PROGRAM P_FastScan
VAR
	ID						:INT:=FastScan;
	SysStep:				DINT;	
	HomeStep:				DINT;	
	RestStep				:DINT;
	MoveStep				:DINT;
	HomeDone:               BOOL;
	FB_move:				FB_MoveFS_Exte;
	FB_home:				FB_Home_X;
	ton_commandtimeout		:TON;

	ton1:Tc2_Standard.TON;	//	命令延迟关闭
	Move_Done				:BOOL;
	NOT_Moving_TimeOut		:BOOL;
	parameter_out_of_range	:BOOL;
	actuator_out_of_pos_range:BOOL;
	actuator_out_of_neg_range:BOOL;	
	homeTimeOut				:BOOL;
	SpeedNotReach			:BOOL;	
	jog_EN					:BOOL;
	ton_Moving				:TON;
	
	direN:BOOL;
	direp:BOOL;
	log_ErrorEnum:Axis_XY_ErrorEnum;
	log_ID:INT;
	i:INT;
	
END_VAR

ACT_LOG();
GVL_API.stAxis[ID].ControlLoopClosed:=Axis[ID].Ref.Status .ControlLoopClosed;

(*****************POS******************************)
GVL_API.stAxis[ID].position:=Axis[ID].Ref.NcToPlc.ActPos;
direN:=Axis[ID].Ref.Status.NegativeDirection;
direp:=Axis[ID].Ref.Status.PositiveDirection;
(*****************SysStep******************************)
CASE SysStep OF
0:	(*wait*)
	_00_Waiting();				
100:(*idle*)		
	_100_Idle();								
200:(*home*)		
	_200_Homing();
300:(*ready*)	
	_300_Ready();							
400:(*disable*)	
	_400_Disable();			
500:(*Moving*)
	_500_Moving();	
600:(*Stopping*)
	_600_Stopping();
700:(*Error*)
	_700_Error();	
800:(*Reset*)
	_800_Reset();		
END_CASE

(*****************Reset*************************)
IF GVL_API.stAxis[ID].reset OR GVL.Reset THEN 
	SysStep:=800;	
END_IF

ACT_SAFETY();


Axis[ID].aReadStatus();
Axis[ID].aReset();

ACTION _00_Waiting:
IF GVL_API.stAxis[ID].initialize THEN 
	GVL_API.stAxis[ID].initialize:=FALSE;
	Axis[ID].aStop(stop_do:=TRUE);
	SysStep:=100;
ELSIF GVL_API.stAxis[ID].homeExe THEN 
	GVL_API.stAxis[ID].homeExe:=FALSE;  
	GVL_API.stAxis[ID].Home_Done:=FALSE;
	SysStep:=200;
ELSIF GVL_API.stAxis[ID].MoveAbsoluteExe OR GVL_API.stAxis[ID].MoveRelativeExe 
		OR GVL_API.stAxis[ID].MoveVelocityExe OR GVL_API.stAxis[ID].JogBackwards 
		OR GVL_API.stAxis[ID].JogForward OR GVL_API.stAxis[ID].MoveConstantVelocity
		OR GVL_API.stAxis[ID].enabled OR GVL_API.stAxis[ID].Disable THEN 
	GVL_API.stAxis[ID].Move_Done:=FALSE;
	SysStep:=300;	
ELSIF GVL_API.stAxis[ID].stop THEN 
	SysStep:=600;	
ELSIF GVL_API.stAxis[ID].reset OR GVL.Reset THEN 
	SysStep:=800;	
END_IF

ton1(IN:=GVL_API.stAxis[ID].Home_Done OR  GVL_API.stAxis[ID].Move_Done , PT:=State_reset_time , Q=> , ET=> );
IF ton1.Q THEN 
	GVL_API.stAxis[ID].Home_Done:=FALSE;
	GVL_API.stAxis[ID].Move_Done:=FALSE;
END_IF
END_ACTION

ACTION _100_Idle:
Axis[ID].aStop(stop_do:=FALSE);
Axis[ID].aPower(power_do:=TRUE);	

IF axis[Id].Ref.Status .ControlLoopClosed THEN 
	GVL_API.stAxis[ID].state:=AxisStateEnum.idle;
	SysStep :=0;
ELSIF GVl.Emstop_Button OR GVL.Emstop_SAFE THEN 
	GVL_API.stAxis[ID].errorid:=Axis_XY_ErrorEnum.emergency_error;
	SysStep:=700;
END_IF

(*******************commandtimeout*********************************)
ton_commandtimeout(IN:=NOT axis[Id].Ref.Status .ControlLoopClosed , 
	PT:=LREAL_TO_TIME(GVL_API.stAxis[ID].commandtimeout*1000) ,
	Q=> , ET=> );
IF ton_commandtimeout.Q  THEN 
	ton_commandtimeout(IN:=FALSE );
	GVL_API.stAxis[ID].errorid:=Axis_XY_ErrorEnum.cmd_timeout;
	SysStep:=700;	
END_IF

(*****************RESET******************************)
IF GVL_API.stAxis[ID].reset OR GVL.HMI_btReset   THEN
	 SysStep:=800;
END_IF
END_ACTION

ACTION _200_Homing:
FB_Home(
		ref:=				Axis[ID].Ref , 
		Execute:= , 
		PosLimit:=			Axis[ID].IO.snLimitP , 
		Position:=			0 , 
		HomeingVelo:=		GVL_API.stAxis[ID].homingvelocity , 
		Standby_position:=  GVL_API.stAxis[ID].homeoffset,
		bCalibrationCam:=	Axis[ID].IO.snHome , 
		rel_dis:=			50 , 
		TimeOutSet:=		GVL_API.stAxis[ID].homingtimeout , 
		reset:= , 
		Done=> , 
		Busy=> , 
		Active=> , 
		CommandAborted=> , 
		Error=> , 
		ErrorID=> , 
		TimeOut=> );
		
CASE HomeStep OF
0:
	IF GVL_API.stAxis[ID].homingvelocity<>0 THEN 
		HomeStep:=10;
	END_IF
10:
	FB_Home.Execute:=TRUE;					
	IF FB_Home.Done THEN
		GVL_API.stAxis[ID].Home_Done:=TRUE;
		FB_Home.Execute:=FALSE;		
		HomeStep:=20;
	END_IF
	IF FB_Home.Error THEN 		
		GVL_API.stAxis[ID].ErrorId:=Axis_XY_ErrorEnum.homing_timeout;
		HomeStep:=30;
	END_IF
	
20:	(**********HOME DONE****************)	
	GVL_API.stAxis[ID].state:=AxisStateEnum.ready;	
	HomeStep:=0;	
	SysStep:=0;
		
30:(**********TIME OUT****************)
	FB_Home.Execute:=FALSE;
	FB_Home.reset:=TRUE;
	HomeStep:=40;
40:(**********RESET****************)
	FB_Home.reset:=FALSE;
	HomeStep:=0;
	SysStep:=700;
		
END_CASE

IF FB_Home.Busy THEN 
	GVL_API.stAxis[ID].state:=AxisStateEnum.homing;
END_IF


(*****************RESET******************************)
IF GVL_API.stAxis[ID].reset    THEN
	FB_Home.Execute:=FALSE;
	 SysStep:=800;
END_IF
END_ACTION

ACTION _300_Ready:
Axis[ID].aStop();
GVL_API.stAxis[ID].Move_Done:=FALSE;
(***********parameter_out_of_range***********)
IF GVL_API.stAxis[ID].requestedposition>GVL_API.stAxis[ID].maxDistance OR GVL_API.stAxis[ID].requestedposition<0 THEN 
		parameter_out_of_range:=TRUE;
ELSIF GVL_API.stAxis[ID].constantvelocitystart>GVL_API.stAxis[ID].maxDistance OR GVL_API.stAxis[ID].constantvelocitystart<0 THEN
		parameter_out_of_range:=TRUE;
ELSIF GVL_API.stAxis[ID].constanvelocityend>GVL_API.stAxis[ID].maxDistance OR GVL_API.stAxis[ID].constanvelocityend<0 THEN
		parameter_out_of_range:=TRUE;	
ELSIF  GVL_API.stAxis[ID].requestedoffset>0 
	AND (GVL_API.stAxis[ID].maxDistance-Axis[ID].Ref.NcToPlc.ActPos)<GVL_API.stAxis[ID].requestedoffset THEN
	 	parameter_out_of_range:=TRUE;
ELSIF GVL_API.stAxis[ID].requestedoffset<-1	
	AND Axis[ID].Ref.NcToPlc.ActPos<ABS(GVL_API.stAxis[ID].requestedoffset) THEN 
		parameter_out_of_range:=TRUE;

ELSE
		parameter_out_of_range:=FALSE;
END_IF	

(*********out_of_pos_range****************)
IF Axis[ID].Ref.NcToPlc.ActPos>GVL_API.stAxis[ID].maxDistance THEN 
	actuator_out_of_pos_range:=TRUE;
	actuator_out_of_neg_range:=FALSE;		
ELSIF	Axis[ID].Ref.NcToPlc.ActPos<-1 THEN 
	actuator_out_of_pos_range:=FALSE;
	actuator_out_of_neg_range:=TRUE;
ELSE
	actuator_out_of_pos_range:=FALSE;
	actuator_out_of_neg_range:=FALSE;
END_IF
	

(*****************state******************************)
IF Axis[ID].Ref.Status.NotMoving AND axis[Id].Ref.Status .ControlLoopClosed  
AND NOT Axis[ID].Ref.Status.Error THEN 
	IF parameter_out_of_range THEN 
		GVL_API.stAxis[ID].errorid:=Axis_XY_ErrorEnum.parameter_out_of_range;
		SysStep:=700;
	ELSIF actuator_out_of_pos_range THEN 
		GVL_API.stAxis[ID].errorid:=Axis_XY_ErrorEnum.actuator_out_of_pos_range;
		SysStep:=700;
	ELSIF actuator_out_of_neg_range THEN 
		GVL_API.stAxis[ID].errorid:=Axis_XY_ErrorEnum.actuator_out_of_neg_range;
		SysStep:=700;	
	ELSE
		GVL_API.stAxis[ID].state:=AxisStateEnum.ready;
		GVL_API.stAxis[ID].errorid:=Axis_XY_ErrorEnum.no_error;
	END_IF
END_IF

(*****************valid command******************************)
IF NOT parameter_out_of_range 
AND axis[Id].Ref.Status .ControlLoopClosed  THEN  			
	IF GVL_API.stAxis[ID].MoveAbsoluteExe OR GVL_API.stAxis[ID].MoveRelativeExe 
		OR GVL_API.stAxis[ID].MoveVelocityExe OR GVL_API.stAxis[ID].JogBackwards 
		OR GVL_API.stAxis[ID].JogForward OR GVL_API.stAxis[ID].MoveConstantVelocity	THEN 	  		
			SysStep:=500;		
	END_IF
END_IF

(*****************enable-disable******************************)
IF GVL_API.stAxis[ID].enabled THEN 
	Axis[Id].aPower(power_do:=TRUE);	
	GVL_API.stAxis[ID].enabled:=FALSE;
	 GVL_API.stAxis[ID].state:=AxisStateEnum.ready;
	SysStep :=0;
ELSIF  GVL_API.stAxis[ID].Disable THEN 
	  SysStep:=400;
END_IF


(*****************RESET******************************)
IF GVL_API.stAxis[ID].reset THEN
	 SysStep:=800;
END_IF
END_ACTION

ACTION _400_Disable:
(*****************enable-disable******************************)
IF GVL_API.stAxis[ID].Disable THEN 
	Axis[Id].aPower(power_do:=FALSE);
	GVL_API.stAxis[ID].Disable:=FALSE;
	GVL_API.stAxis[ID].state:=AxisStateEnum.disabled;
	//IF NOT  axis[Id].Ref.Status .ControlLoopClosed THEN 
		SysStep:=0;
	//END_IF
	
END_IF

(*****************RESET******************************)
IF GVL_API.stAxis[ID].reset THEN
	 SysStep:=800;
END_IF
END_ACTION

ACTION _500_Moving:
GVL_API.stAxis[ID].state:=AxisStateEnum.moving;

(*********out_of_pos_range****************)
IF Axis[ID].Ref.NcToPlc.ActPos>GVL_API.stAxis[ID].maxDistance THEN 
	actuator_out_of_pos_range:=TRUE;
	actuator_out_of_neg_range:=FALSE;
	GVL_API.stAxis[ID].JogForward:=FALSE;		
ELSIF	Axis[ID].Ref.NcToPlc.ActPos<-1 THEN 
	actuator_out_of_pos_range:=FALSE;
	actuator_out_of_neg_range:=TRUE;
	GVL_API.stAxis[ID].JogBackwards:=FALSE;
ELSE
	actuator_out_of_pos_range:=FALSE;
	actuator_out_of_neg_range:=FALSE;
END_IF

(*********parameter_out_of_range****************)
IF Axis[ID].IO.snHome 
	AND (GVL_API.stAxis[ID].requestedoffset<0 
	OR GVL_API.stAxis[ID].constantvelocitystart<Axis[ID].Ref.NcToPlc.ActPos
	OR GVL_API.stAxis[ID].constanvelocityend<Axis[ID].Ref.NcToPlc.ActPos
	OR GVL_API.stAxis[ID].requestedposition<Axis[ID].Ref.NcToPlc.ActPos)
	THEN 	parameter_out_of_range:=TRUE;
ELSIF Axis[ID].IO.snLimitP
	AND (GVL_API.stAxis[ID].requestedoffset>0 
	OR GVL_API.stAxis[ID].constantvelocitystart>Axis[ID].Ref.NcToPlc.ActPos
	OR GVL_API.stAxis[ID].constanvelocityend>Axis[ID].Ref.NcToPlc.ActPos
	OR GVL_API.stAxis[ID].requestedposition>Axis[ID].Ref.NcToPlc.ActPos)
	THEN 	parameter_out_of_range:=TRUE;
END_IF


IF NOT_Moving_TimeOut OR GVL_API.stAxis[ID].Move_Done  THEN 			(************NOT_Moving_TimeOut/Move_Done**************)
	NOT_Moving_TimeOut:=FALSE;	
	GVL_API.stAxis[ID].state:=AxisStateEnum.ready;			
	SysStep:=0;
ELSIF SpeedNotReach THEN 							(************SpeedNotReach**************)
	GVL_API.stAxis[ID].errorid:=Axis_XY_ErrorEnum.SpeedNotReach;
	SysStep:=700;
ELSIF Axis[ID].Ref.Status.NotMoving AND parameter_out_of_range THEN 
	GVL_API.stAxis[ID].errorid:=Axis_XY_ErrorEnum.parameter_out_of_range;
	SysStep:=700;
ELSIF Axis[ID].Ref.Status.Moving THEN 				(************trigger_limit**************)
	IF (Axis[ID].Ref.Status.NegativeDirection AND Axis[ID].IO.snLimitN) OR 
		(Axis[ID].Ref.Status.PositiveDirection AND Axis[ID].IO.snLimitP) 
		OR stInput.biElectromagnet_limit  OR stOutput.bqElectromagnet_power 
	THEN	
		Axis[ID].aStop(stop_do:=TRUE);
		GVL_API.stAxis[ID].errorid:=Axis_XY_ErrorEnum.trigger_limit;
		SysStep:=700;	
	END_IF 
	
ELSIF actuator_out_of_pos_range THEN 					(*********out_of_pos_range****************)
	Axis[ID].aStop(stop_do:=TRUE);
	GVL_API.stAxis[ID].errorid:=Axis_XY_ErrorEnum.actuator_out_of_pos_range;
	SysStep:=700;
ELSIF actuator_out_of_neg_range THEN
	Axis[ID].aStop(stop_do:=TRUE); 
	GVL_API.stAxis[ID].errorid:=Axis_XY_ErrorEnum.actuator_out_of_neg_range;
	SysStep:=700;	
ELSE GVL_API.stAxis[ID].errorid:=Axis_XY_ErrorEnum.no_error;
END_IF


(*****************JOG/ABS/REL/******************************)
(*****************MoveConstantVelocity*****************************)
IF NOT parameter_out_of_range  THEN 
	FB_move(
	enable:= 					NOT stInput.biElectromagnet_limit AND NOT stOutput.bqElectromagnet_power,	
	ref:= 						Axis[ID].Ref, 
	jogF:= 						GVL_API.stAxis[ID].JogForward, 
	jogB:= 						GVL_API.stAxis[ID].JogBackwards, 
	Move_Stop:=				GVL_API.stAxis[ID].stop OR GVL_API.stAxis[ID].reset ,
	PosLimit:=					Axis[ID].IO.snLimitP , 
	NegLimit:= 					Axis[ID].IO.snLimitN, 
	maxDistance:=				GVL_API.stAxis[ID].maxDistance ,	
	Acceleration:= 				GVL_API.stAxis[ID].acceleration, 
	Deceleration:= 				GVL_API.stAxis[ID].acceleration, 
	Jerk:= 						GVL_API.stAxis[ID].jerk, 	 
	MoveRelExe:= 				GVL_API.stAxis[ID].MoveRelativeExe, 
	MoveAbsExe:= 				GVL_API.stAxis[ID].MoveAbsoluteExe, 
	MoveConstantVelocityExe:= 	GVL_API.stAxis[ID].MoveConstantVelocity, 
	Velo:= 						GVL_API.stAxis[ID].velocity, 
	TargetRel:= 				GVL_API.stAxis[ID].requestedoffset, 
	TargetAbs:= 				GVL_API.stAxis[ID].requestedposition, 
	constantvelocitystart:= 	GVL_API.stAxis[ID].constantvelocitystart, 
	constanvelocityend:= 		GVL_API.stAxis[ID].constanvelocityend, 
	Done:= 						GVL_API.stAxis[ID].Move_Done,
	NotMovingTimeOut:= 			NOT_Moving_TimeOut,
	SpeedNotReach:=				SpeedNotReach
	);	
END_IF


(*****************stop******************************)
IF GVL_API.stAxis[ID].stop THEN 
	SysStep:=600;
END_IF
(*****************RESET******************************)
IF GVL_API.stAxis[ID].reset THEN
	 SysStep:=800;
END_IF
END_ACTION

ACTION _600_Stopping:
(**************只单独用作STOP命令*************************)
GVL_API.stAxis[ID].state:=AxisStateEnum.stopping;

Axis[ID].aStop(stop_do:=GVL_API.stAxis[ID].stop,Jerk:=GVL_API.stAxis[ID].jerk);
IF Axis[ID].mcStop.Busy THEN 
	GVL_API.stAxis[ID].state:=AxisStateEnum.stopping;	
	GVL_API.stAxis[ID].JogBackwards:=FALSE;
	GVL_API.stAxis[ID].JogForward:=FALSE;
	GVL_API.stAxis[ID].MoveAbsoluteExe:=FALSE;
	GVL_API.stAxis[ID].MoveConstantVelocity:=FALSE;
	GVL_API.stAxis[ID].MoveRelativeExe:=FALSE;
	GVL_API.stAxis[ID].velocity:=0;
	GVL_API.stAxis[ID].requestedoffset:=0;
	GVL_API.stAxis[ID].requestedposition:=0;
	GVL_API.stAxis[ID].stop:=FALSE;
END_IF

IF Axis[ID].mcStop.Done AND Axis[ID].Ref.Status.NotMoving   THEN 		
	GVL_API.stAxis[ID].stop:=FALSE;
	GVL_API.stAxis[ID].state:=AxisStateEnum.ready;	
	GVL_API.stAxis[ID].Move_Done:=TRUE;
	SysStep:=0;
END_IF

(*****************RESET******************************)
IF GVL_API.stAxis[ID].reset THEN
	 GVL_API.stAxis[ID].stop:=FALSE;
	 Axis[ID].aStop(stop_do:=FALSE);
	 SysStep:=800;
END_IF
END_ACTION

ACTION _700_Error:
(*****************ERROR******************************)
GVL_API.stAxis[ID].Error:=TRUE;
GVL_API.stAxis[ID].state:=AxisStateEnum.error;
		GVL_API.stAxis[ID].initialize:=FALSE;
		GVL_API.stAxis[ID].homeExe:=FALSE; 
		GVL_API.stAxis[ID].stop:=FALSE;
		GVL_API.stAxis[ID].JogBackwards:=FALSE;
		GVL_API.stAxis[ID].JogForward:=FALSE;
		GVL_API.stAxis[ID].MoveAbsoluteExe:=FALSE;
		GVL_API.stAxis[ID].MoveConstantVelocity:=FALSE;
		GVL_API.stAxis[ID].MoveRelativeExe:=FALSE;
		GVL_API.stAxis[ID].velocity:=0;
		GVL_API.stAxis[ID].requestedoffset:=0;
		GVL_API.stAxis[ID].requestedposition:=0;
		GVL_API.stAxis[ID].constantvelocitystart:=0;
		GVL_API.stAxis[ID].constanvelocityend:=0;
		FB_Home.Execute:=FALSE;
		GVL_API.stAxis[ID].Home_Done:=FALSE;
		GVL_API.stAxis[ID].Move_Done:=FALSE;
 SysStep:=0;
END_ACTION

ACTION _800_Reset:
Axis[ID].aStop();
CASE RestStep OF
0:(***************复位命令**************************)
	IF GVL_API.stAxis[ID].reset OR GVL.Reset THEN
		GVL_API.stAxis[ID].initialize:=FALSE;
		GVL_API.stAxis[ID].homeExe:=FALSE; 
		GVL_API.stAxis[ID].stop:=FALSE;
		GVL_API.stAxis[ID].JogBackwards:=FALSE;
		GVL_API.stAxis[ID].JogForward:=FALSE;
		GVL_API.stAxis[ID].MoveAbsoluteExe:=FALSE;
		GVL_API.stAxis[ID].MoveConstantVelocity:=FALSE;
		GVL_API.stAxis[ID].MoveRelativeExe:=FALSE;
		GVL_API.stAxis[ID].velocity:=0;
		GVL_API.stAxis[ID].requestedoffset:=0;
		GVL_API.stAxis[ID].requestedposition:=0;
		GVL_API.stAxis[ID].constantvelocitystart:=0;
		GVL_API.stAxis[ID].constanvelocityend:=0;
		FB_Home(ref:=Axis[ID].Ref , Execute:= FALSE);
		GVL_API.stAxis[ID].Home_Done:=FALSE;
		GVL_API.stAxis[ID].Move_Done:=FALSE;
		RestStep:=1;
	END_IF
1:	
		RestStep:=2;

2:(***************EORROR来的错误**************************)
		GVL_API.stAxis[ID].reset:=FALSE;
		parameter_out_of_range:=FALSE;
		SpeedNotReach:=FALSE;		
		RestStep:=20;
	
10:	(***************轴错误复位**************************)		
		Axis[ID].Reset_do:=TRUE;		
		RestStep:=100;		
20:	(***************轴停止*****************************)
		Axis[ID].aStop(stop_do:=TRUE);		
		RestStep:=30;
30:
	IF  Axis[ID].Ref.Status.NotMoving   THEN 		
		RestStep:=10;	
	END_IF
100:		
	IF Axis[ID].Ref.Status.NotMoving THEN 
		Axis[Id].aPower(power_do:=FALSE);
		GVL_API.stAxis[ID].Error:=FALSE;
		GVL_API.stAxis[ID].state:=AxisStateEnum.off;
		GVL_API.stAxis[ID].Errorid:=Axis_XY_ErrorEnum.no_error;
			SysStep:=0;
			RestStep:=0;
	END_IF
	  
END_CASE
END_ACTION

ACTION ACT_LOG:
(*************************LOG*******************************************)
log_ID:=100;
//initialize
AlarmActionArray[log_ID+1].AlarmMsg.EN	:=	'Fast Scan Initialize cmdtimeout:';
AlarmActionArray[log_ID+1].AlarmMsg.EN	:=CONCAT(AlarmActionArray[log_ID+1].AlarmMsg.EN,
																	LREAL_TO_STRING(GVL_API.stAxis[ID].commandtimeout));
AlarmActionArray[log_ID+1].AlarmMsg.EN	:=CONCAT(AlarmActionArray[log_ID+1].AlarmMsg.EN,'; velocity:');
AlarmActionArray[log_ID+1].AlarmMsg.EN	:=CONCAT(AlarmActionArray[log_ID+1].AlarmMsg.EN,
																	LREAL_TO_STRING(GVL_API.stAxis[ID].velocity));	
AlarmActionArray[log_ID+1].AlarmMsg.EN	:=CONCAT(AlarmActionArray[log_ID+1].AlarmMsg.EN,'; acce:');																
AlarmActionArray[log_ID+1].AlarmMsg.EN	:=CONCAT(AlarmActionArray[log_ID+1].AlarmMsg.EN,
																	LREAL_TO_STRING(GVL_API.stAxis[ID].acceleration));
AlarmActionArray[log_ID+1].AlarmMsg.EN	:=CONCAT(AlarmActionArray[log_ID+1].AlarmMsg.EN,'; maxposition:');	
AlarmActionArray[log_ID+1].AlarmMsg.EN	:=CONCAT(AlarmActionArray[log_ID+1].AlarmMsg.EN,
																	LREAL_TO_STRING(GVL_API.stAxis[ID].maxDistance));
fbSetAlarm[log_ID+1](
	InUse:=TRUE , 
	//EventId:=log_ID+1 , 
	EventActive:=GVL_API.stAxis[ID].initialize , 
	EventClass:=Alm_EventClass.Event , 
	ToTheLogFile:=TRUE, 
	ToTheHistory:=TRUE , 
 );
 //home
AlarmActionArray[log_ID+2].AlarmMsg.EN	:=	'Fast Scan Home homingvelocity:';
AlarmActionArray[log_ID+2].AlarmMsg.EN	:=CONCAT(AlarmActionArray[log_ID+2].AlarmMsg.EN,
																	LREAL_TO_STRING(GVL_API.stAxis[ID].homingvelocity));
AlarmActionArray[log_ID+2].AlarmMsg.EN	:=CONCAT(AlarmActionArray[log_ID+2].AlarmMsg.EN,'; homeoffset:');
AlarmActionArray[log_ID+2].AlarmMsg.EN	:=CONCAT(AlarmActionArray[log_ID+2].AlarmMsg.EN,
																	LREAL_TO_STRING(GVL_API.stAxis[ID].homeoffset));		
AlarmActionArray[log_ID+2].AlarmMsg.EN	:=CONCAT(AlarmActionArray[log_ID+2].AlarmMsg.EN,'; homingtimeout:');
AlarmActionArray[log_ID+2].AlarmMsg.EN	:=CONCAT(AlarmActionArray[log_ID+2].AlarmMsg.EN,
																	LREAL_TO_STRING(GVL_API.stAxis[ID].homingtimeout));																
fbSetAlarm[log_ID+2](
	InUse:=TRUE , 
	//EventId:=log_ID+2 , 
	EventActive:=GVL_API.stAxis[ID].homeExe , 
	EventClass:=Alm_EventClass.Event , 
	ToTheLogFile:=TRUE, 
	ToTheHistory:=TRUE , 
 );
 //MoveRelative
AlarmActionArray[log_ID+3].AlarmMsg.EN	:=CONCAT('Fast Scan MoveRelative displacement:',
																	LREAL_TO_STRING(GVL_API.stAxis[ID].requestedoffset));
AlarmActionArray[log_ID+3].AlarmMsg.EN	:=CONCAT(AlarmActionArray[log_ID+3].AlarmMsg.EN,'; velocity:');
AlarmActionArray[log_ID+3].AlarmMsg.EN	:=CONCAT(AlarmActionArray[log_ID+3].AlarmMsg.EN,
																	LREAL_TO_STRING(GVL_API.stAxis[ID].velocity));
AlarmActionArray[log_ID+3].AlarmMsg.EN	:=CONCAT(AlarmActionArray[log_ID+3].AlarmMsg.EN,'; acc:');
AlarmActionArray[log_ID+3].AlarmMsg.EN	:=CONCAT(AlarmActionArray[log_ID+3].AlarmMsg.EN,
																	LREAL_TO_STRING(GVL_API.stAxis[ID].acceleration));
AlarmActionArray[log_ID+3].AlarmMsg.EN	:=CONCAT(AlarmActionArray[log_ID+3].AlarmMsg.EN,'; jerk:');																	
AlarmActionArray[log_ID+3].AlarmMsg.EN	:=CONCAT(AlarmActionArray[log_ID+3].AlarmMsg.EN,
																	LREAL_TO_STRING(GVL_API.stAxis[ID].jerk));
fbSetAlarm[log_ID+3](
	InUse:=TRUE , 
	//EventId:=log_ID+3 , 
	EventActive:=GVL_API.stAxis[ID].MoveRelativeExe , 
	EventClass:=Alm_EventClass.Event , 
	ToTheLogFile:=TRUE, 
	ToTheHistory:=TRUE , 
 );
 //MoveAbsoluteExe
AlarmActionArray[log_ID+4].AlarmMsg.EN	:=CONCAT('Fast Scan MoveAbsolute position:',
																	LREAL_TO_STRING(GVL_API.stAxis[ID].requestedposition));
AlarmActionArray[log_ID+4].AlarmMsg.EN	:=CONCAT(AlarmActionArray[log_ID+4].AlarmMsg.EN,'; velocity:');
AlarmActionArray[log_ID+4].AlarmMsg.EN	:=CONCAT(AlarmActionArray[log_ID+4].AlarmMsg.EN,
																	LREAL_TO_STRING(GVL_API.stAxis[ID].velocity));
AlarmActionArray[log_ID+4].AlarmMsg.EN	:=CONCAT(AlarmActionArray[log_ID+4].AlarmMsg.EN,'; acc:');
AlarmActionArray[log_ID+4].AlarmMsg.EN	:=CONCAT(AlarmActionArray[log_ID+4].AlarmMsg.EN,
																	LREAL_TO_STRING(GVL_API.stAxis[ID].acceleration));
AlarmActionArray[log_ID+4].AlarmMsg.EN	:=CONCAT(AlarmActionArray[log_ID+4].AlarmMsg.EN,'; jerk:');																	
AlarmActionArray[log_ID+4].AlarmMsg.EN	:=CONCAT(AlarmActionArray[log_ID+4].AlarmMsg.EN,
																	LREAL_TO_STRING(GVL_API.stAxis[ID].jerk));
fbSetAlarm[log_ID+4](
	InUse:=TRUE , 
	//EventId:=log_ID+4 , 
	EventActive:=GVL_API.stAxis[ID].MoveAbsoluteExe , 
	EventClass:=Alm_EventClass.Event , 
	ToTheLogFile:=TRUE, 
	ToTheHistory:=TRUE , 
 );
 //MoveConstantVelocity
AlarmActionArray[log_ID+5].AlarmMsg.EN	:=CONCAT('Fast Scan MoveConstantVelocity,',
																LREAL_TO_STRING(GVL_API.stAxis[ID].constantvelocitystart));
AlarmActionArray[log_ID+5].AlarmMsg.EN	:=CONCAT(AlarmActionArray[log_ID+5].AlarmMsg.EN,'->');
AlarmActionArray[log_ID+5].AlarmMsg.EN	:=CONCAT(AlarmActionArray[log_ID+5].AlarmMsg.EN,
																LREAL_TO_STRING(GVL_API.stAxis[ID].constanvelocityend));
AlarmActionArray[log_ID+5].AlarmMsg.EN	:=CONCAT(AlarmActionArray[log_ID+5].AlarmMsg.EN,'->');
AlarmActionArray[log_ID+5].AlarmMsg.EN	:=CONCAT(AlarmActionArray[log_ID+5].AlarmMsg.EN,
																LREAL_TO_STRING(GVL_API.stAxis[ID].requestedposition));
AlarmActionArray[log_ID+5].AlarmMsg.EN	:=CONCAT(AlarmActionArray[log_ID+5].AlarmMsg.EN,'; velocity:');
AlarmActionArray[log_ID+5].AlarmMsg.EN	:=CONCAT(AlarmActionArray[log_ID+5].AlarmMsg.EN,
																	LREAL_TO_STRING(GVL_API.stAxis[ID].velocity));
AlarmActionArray[log_ID+5].AlarmMsg.EN	:=CONCAT(AlarmActionArray[log_ID+5].AlarmMsg.EN,'; acc:');
AlarmActionArray[log_ID+5].AlarmMsg.EN	:=CONCAT(AlarmActionArray[log_ID+5].AlarmMsg.EN,
																	LREAL_TO_STRING(GVL_API.stAxis[ID].acceleration));
AlarmActionArray[log_ID+5].AlarmMsg.EN	:=CONCAT(AlarmActionArray[log_ID+5].AlarmMsg.EN,'; jerk:');																	
AlarmActionArray[log_ID+5].AlarmMsg.EN	:=CONCAT(AlarmActionArray[log_ID+5].AlarmMsg.EN,
																	LREAL_TO_STRING(GVL_API.stAxis[ID].jerk));
fbSetAlarm[log_ID+5](
	InUse:=TRUE , 
	//EventId:=log_ID+5 , 
	EventActive:=GVL_API.stAxis[ID].MoveConstantVelocity , 
	EventClass:=Alm_EventClass.Event , 
	ToTheLogFile:=TRUE, 
	ToTheHistory:=TRUE , 
 );
//stop
AlarmActionArray[log_ID+6].AlarmMsg.EN	:=	'Fast Scan MoveStop ';
fbSetAlarm[log_ID+6](
	InUse:=TRUE , 
	//EventId:=log_ID+6 , 
	EventActive:=GVL_API.stAxis[ID].stop , 
	EventClass:=Alm_EventClass.Event , 
	ToTheLogFile:=TRUE, 
	ToTheHistory:=TRUE , 
 );
 //enabled
AlarmActionArray[log_ID+7].AlarmMsg.EN	:=	'Fast Scan Enabled ';
fbSetAlarm[log_ID+7](
	InUse:=TRUE , 
	//EventId:=log_ID+7 , 
	EventActive:=GVL_API.stAxis[ID].enabled , 
	EventClass:=Alm_EventClass.Event , 
	ToTheLogFile:=TRUE, 
	ToTheHistory:=TRUE , 
 );
  //disable
AlarmActionArray[log_ID+8].AlarmMsg.EN	:=	'Fast Scan Disable ';
fbSetAlarm[log_ID+8](
	InUse:=TRUE , 
	//EventId:=log_ID+8 , 
	EventActive:=GVL_API.stAxis[ID].Disable , 
	EventClass:=Alm_EventClass.Event , 
	ToTheLogFile:=TRUE, 
	ToTheHistory:=TRUE , 
 );
//ERROR,log_ErrorEnum只能等于一个常数
CASE GVL_API.stAxis[ID].errorid  OF
0	:	log_ErrorEnum	:=	0	;
1	:	log_ErrorEnum	:=	1	;
2	:	log_ErrorEnum	:=	2	;
3	:	log_ErrorEnum	:=	3	;
4	:	log_ErrorEnum	:=	4	;
5	:	log_ErrorEnum	:=	5	;
6	:	log_ErrorEnum	:=	6	;
7	:	log_ErrorEnum	:=	7	;
8	:	log_ErrorEnum	:=	8	;
9	:	log_ErrorEnum	:=	9	;
10	:	log_ErrorEnum	:=	10	;
11	:	log_ErrorEnum	:=	11	;
12	:	log_ErrorEnum	:=	12	;
13	:	log_ErrorEnum	:=	13	;
14	:	log_ErrorEnum	:=	14	;
15	:	log_ErrorEnum	:=	15	;
16	:	log_ErrorEnum	:=	16	;
666	:	log_ErrorEnum	:=	666	;

END_CASE

AlarmActionArray[log_ID+9].AlarmMsg.EN	:=CONCAT('Fast Scan Error: ',TO_STRING(log_ErrorEnum));
fbSetAlarm[log_ID+9](
	InUse:=TRUE , 
//	EventId:=log_ID+9 , 
	EventActive:=GVL_API.stAxis[ID].errorid<>0 AND GVL_API.stAxis[ID].errorid<>666 , 
	EventClass:=Alm_EventClass.Alarm , 
	ToTheLogFile:=TRUE, 
	ToTheHistory:=TRUE , 
 );
 
//reset
AlarmActionArray[log_ID+10].AlarmMsg.EN	:=	'Fast Scan Reset ';
fbSetAlarm[log_ID+10](
	InUse:=TRUE , 
	EventId:=log_ID+10 , 
	EventActive:=GVL_API.stAxis[ID].reset , 
	EventClass:=Alm_EventClass.Event , 
	ToTheLogFile:=TRUE, 
	ToTheHistory:=TRUE , 
 );
 //AXIX_ERRORID
 AlarmActionArray[log_ID+11].AlarmMsg.EN	:=CONCAT('Fast Scan Axis_ErrorID: ',
																		UDINT_TO_STRING(Axis[ID].Ref.Status.ErrorID));
fbSetAlarm[log_ID+11](
	InUse:=TRUE , 
	EventId:=log_ID+11 , 
	EventActive:=Axis[ID].Ref.Status.Error , 
	EventClass:=Alm_EventClass.Event , 
	ToTheLogFile:=TRUE, 
	ToTheHistory:=TRUE , 
 );
END_ACTION

ACTION ACT_Safety:
(*****************SAFETY******************************)
IF GVL_API.stAxis[ID].state<>AxisStateEnum.off AND  GVL_API.stAxis[ID].state<>AxisStateEnum.error THEN 
	IF GVl.Emstop_Button OR GVL.Emstop_SAFE  THEN 
		GVL_API.stAxis[ID].errorid:=Axis_XY_ErrorEnum.emergency_error;
		Axis[ID].aStop(stop_do:=TRUE,Dec:=HMI_EM_STOP_Dec_FS,Jerk:=HMI_EM_STOP_Jerk_FS);
		//Axis[ID].aStop(stop_do:=TRUE,Jerk:=GVL_API.stAxis[ID].jerk);
		SysStep:=700;
	ELSIF GVL.shuttle_crash OR  Axis[ID].IO.snLimitN OR Axis[ID].IO.snLimitP  THEN 	
		GVL_API.stAxis[ID].errorid:=Axis_XY_ErrorEnum.trigger_Limit;
		Axis[ID].aStop(stop_do:=TRUE,Dec:=HMI_EM_STOP_Dec_FS,Jerk:=HMI_EM_STOP_Jerk_FS);
		SysStep:=700;
	(*ELSIF GVL.interlock_triggered THEN 
		GVL_API.stAxis[ID].ErrorId:=Axis_XY_ErrorEnum.interlock_error;
		Axis[ID].aStop(stop_do:=TRUE,Dec:=HMI_EM_STOP_Dec_FS,Jerk:=HMI_EM_STOP_Jerk_FS);
		SysStep:=700;
	*)
	ELSIF  Axis[ID].mcReadStatus.ErrorID=18000 THEN 
		GVL_API.stAxis[ID].errorid:=Axis_XY_ErrorEnum.Drive_not_ready_for_operation;
		SysStep:=700;
	ELSIF   Axis[ID].mcReadStatus.ErrorID=17510 THEN 
		GVL_API.stAxis[ID].errorid:=Axis_XY_ErrorEnum.Invalid_IO_data_for_more_than_n_subsequent_NC_cycles_encoder;
		SysStep:=700;	
	ELSIF  Axis[ID].mcReadStatus.ErrorID<>0 THEN 
		GVL_API.stAxis[ID].errorid:=Axis[ID].mcReadStatus.ErrorID;
		SysStep:=700;
	//ELSE 
	//	GVL_API.stAxis[ID].error:=Axis_XY_ErrorEnum.no_error;
	//	SysStep:=700;			
	END_IF	
END_IF

(*****************AXIS_ERROR******************************)
GVL_API.stAxis[ID].AxisErrorId:=Axis[ID].Ref.Status.ErrorID;
END_ACTION

END_PROGRAM

(* stored: Version 1.1.0.1, ProductVersion 3.1.4024.11
   POU P_FastScan: Id {7cc9c2b1-b180-471a-b758-cdc159abd7da}, SpecialFunc None
   Folder SysStep: Id {a63258c5-3aed-4796-800f-5a36c19be8da}
   Action _00_Waiting: Id {9769fe14-e4b9-4259-b6f0-64c972a63d61}
   Action _100_Idle: Id {5480bc58-5b5a-422f-9895-895a095013f1}
   Action _200_Homing: Id {ff145943-35b0-4af2-b6a1-94645a607907}
   Action _300_Ready: Id {6d9bf504-d754-4d3d-8e99-a60116d2aa64}
   Action _400_Disable: Id {4591e4a3-1e6c-4f02-aa39-b0aa5f548b78}
   Action _500_Moving: Id {fece1bfa-205f-44d0-baf5-fde7e70c7241}
   Action _600_Stopping: Id {9569bd56-b8fd-434a-826a-0242c0f97c20}
   Action _700_Error: Id {74fba152-571e-44d0-b38a-4cabe217ad6d}
   Action _800_Reset: Id {60ece19a-2d3c-4abc-8107-c7a66e6ddb1d}
   Action ACT_LOG: Id {a430402b-6307-44b3-8d4d-23cfdb5d6666}
   Action ACT_Safety: Id {76dcdea7-03b4-40e5-8999-5c191b7963bc} *)
